(* Logix 5000 project; controller Injection_Comorfords vendor 1 type 14 code 222 rev 33.11; software revision 33.00 *)

TASK MainTask (continuous, watchdog 500 ms) : MainProgram
TASK SafetyTask (periodic, rate 20 ms, priority 10, watchdog 20 ms, safety) : SafetyProgram

MODULES
   Local : vendor 1 type 14 code 222 (5069 0, rev 33.11)
      WTU_C1_C2 : vendor 1 type 0 code 23 (Ethernet 192.168.2.12, rev 1.1)   // water tempering unit PLC
      WTU_C3_C4 : vendor 1 type 0 code 23 (Ethernet 192.168.2.13, rev 1.1)   // water tempering unit PLC
      PF525_Stirrer_Tank_1 : PowerFlex 525-EENET (Ethernet 192.168.2.15, rev 5.2, Output RPI 20 ms)   // 0.75 kW
      PF525_Feedingpump_1 : PowerFlex 525-EENET (Ethernet 192.168.2.16, rev 5.2, Output RPI 20 ms)   // 0.75 kW
      PF525_CIP_Pump_1 : PowerFlex 525-EENET (Ethernet 192.168.2.17, rev 5.2, Output RPI 20 ms)   // 0.75 kW
      PF525_Stirrer_Tank_2 : PowerFlex 525-EENET (Ethernet 192.168.2.18, rev 5.2, Output RPI 20 ms)   // 0.75 kW
      PF525_Feedingpump_2 : PowerFlex 525-EENET (Ethernet 192.168.2.19, rev 5.2, Output RPI 20 ms)   // 0.75 kW
      PF525_CIP_Pump_2 : PowerFlex 525-EENET (Ethernet 192.168.2.20, rev 5.2, Output RPI 20 ms)   // 0.75 kW
      Manifold_Cream : 2198-H008-ERS2 (Ethernet 192.168.2.22, rev 7.1, AMotionDiagnostics RPI 1 ms, CSafety_Output RPI 20 ms, DSafety_Input RPI 10 ms)
      Manifold_Jam : 2198-H008-ERS2 (Ethernet 192.168.2.23, rev 7.1, AMotionDiagnostics RPI 1 ms, CSafety_Output RPI 20 ms, DSafety_Input RPI 10 ms)
      X_Axis : 2198-H008-ERS2 (Ethernet 192.168.2.24, rev 7.1, AMotionDiagnostics RPI 1 ms, CSafety_Output RPI 20 ms, DSafety_Input RPI 10 ms)
      Z_Axis : 2198-H008-ERS2 (Ethernet 192.168.2.25, rev 7.1, AMotionDiagnostics RPI 1 ms, CSafety_Output RPI 20 ms, DSafety_Input RPI 10 ms)
      U2_MCC1_IO : 1734-AENTR (Ethernet 192.168.2.14, rev 6.1, Output RPI 20 ms)
         U2_MCC1_DIG_In_1 : 1734-IB8 (PointIO 3, rev 3.1)
         U2_MCC1_DIG_In_2 : 1734-IB8 (PointIO 4, rev 3.1)
         U2_MCC1_DIG_In_3 : 1734-IB8 (PointIO 5, rev 3.1)
         U2_MCC1_ANA_In_1 : vendor 1 type 115 code 210 (PointIO 6, rev 3.1, Input RPI 80 ms)
         U2_MCC1_DIG_Out_1 : vendor 1 type 7 code 231 (PointIO 7, rev 3.1)
         U2_MCC1_DIG_Out_2 : vendor 1 type 7 code 231 (PointIO 8, rev 3.1)
         U2_MCC1_DIG_Out_3 : 1734-OB8 (PointIO 9, rev 3.1)
         U2_MCC1_DIG_Out_4 : 1734-OB8 (PointIO 10, rev 3.1)
         U2_MCC1_DIG_Out_5 : 1734-OB8 (PointIO 11, rev 3.1)
         U2_MCC1_DIG_Out_6 : 1734-OB8 (PointIO 12, rev 3.1)
         U2_MCC1_Safety_DIG_In_1 : vendor 1 type 35 code 15 (PointIO 1, rev 2.1, Input RPI 10 ms, Output RPI 20 ms)
         U2_MCC1_Safety_DIG_Out_1 : vendor 1 type 35 code 16 (PointIO 2, rev 2.1, Input RPI 10 ms, Output RPI 20 ms)
      U5_MCC1_IO : 1734-AENTR (Ethernet 192.168.2.21, rev 6.1, Output RPI 20 ms)
         U5_MC1_DIG_In_1 : 1734-IB8 (PointIO 3, rev 3.1)
         U5_MC1_DIG_In_2 : 1734-IB8 (PointIO 4, rev 3.1)
         U5_MC1_DIG_In_3 : 1734-IB8 (PointIO 5, rev 3.1)
         U5_MC1_ANA_In_1 : 1734-IE4C (PointIO 6, rev 3.1, Input RPI 80 ms)
         U5_MC1_ANA_In_2 : 1734-IE4C (PointIO 7, rev 3.1, Input RPI 80 ms)
         U5_MC1_DIG_Out_1 : vendor 1 type 7 code 231 (PointIO 8, rev 3.1)
         U5_MC1_DIG_Out_2 : vendor 1 type 7 code 231 (PointIO 9, rev 3.1)
         U5_MC1_DIG_Out_3 : vendor 1 type 7 code 231 (PointIO 10, rev 3.1)
         U5_MC1_ANA_Out_1 : 1734-OE2C (PointIO 11, rev 3.1, Output RPI 80 ms)
         U5_MC1_Safety_DIG_Out_1 : vendor 1 type 35 code 16 (PointIO 2, rev 2.1, Output RPI 20 ms, Input RPI 10 ms)
         U5_MC1_Safety_DIG_In_1 : vendor 1 type 35 code 15 (PointIO 1, rev 2.1, Input RPI 10 ms, Output RPI 20 ms)
END_MODULES

PROGRAM MainProgram   (* main routine MainRoutine *)

ROUTINE MainRoutine   (* ladder *)
END_ROUTINE
END_PROGRAM

PROGRAM SafetyProgram   (* main routine MainRoutine, safety *)

ROUTINE MainRoutine   (* ladder *)
END_ROUTINE
END_PROGRAM
